FUNCTION_BLOCK Linearachse
VAR_INPUT
END_VAR
VAR_OUTPUT
END_VAR
VAR
END_VAR

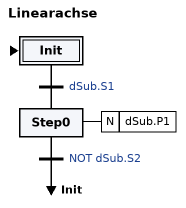
INITIAL_STEP Init:
END_STEP
TRANSITION FROM Init TO Step0
    := dSub.S1;
END_TRANSITION
STEP Step0:
    dSub.P1(N);
END_STEP
TRANSITION FROM Step0 TO Init
    := NOT dSub.S2;
END_TRANSITION

END_FUNCTION_BLOCK

(* stored: Version 1.1.0.1, ProductVersion 3.1.4022.6
   POU Linearachse: Id {aea3de1b-05a0-4fca-a6ab-4cf670639743}, SpecialFunc None *)
